// TIA Portal project "Process" (V16)

(* hardware
DEVICE "S7-1200 station_1"  S7-1200 Station
   slot 0: "Rack_0"  S7-1200 Rack  Rack  V1.0
   slot 1: "PLC_1"  CPU 1212C DC/DC/DC  6ES7 212-1AE40-0XB0  V4.4
   slot 2: "DI 8/DQ 8x24VDC_1"  6ES7 223-1BH32-0XB0  V2.0
   slot 3: "AI 4x13BIT/AQ 2x14BIT_1"  6ES7 234-4HE32-0XB0  V2.1
*)

// ===== PLC "PLC_1"  CPU 1212C DC/DC/DC =====

VAR_GLOBAL   // PLC tag table "Default tag table"
   "System_Byte" AT %MB1 : Byte;
   "FirstScan" AT %M1.0 : Bool;
   "DiagStatusUpdate" AT %M1.1 : Bool;
   "AlwaysTRUE" AT %M1.2 : Bool;
   "AlwaysFALSE" AT %M1.3 : Bool;
   "Clock_Byte" AT %MB0 : Byte;
   "Clock_10Hz" AT %M0.0 : Bool;
   "Clock_5Hz" AT %M0.1 : Bool;
   "Clock_2.5Hz" AT %M0.2 : Bool;
   "Clock_2Hz" AT %M0.3 : Bool;
   "Clock_1.25Hz" AT %M0.4 : Bool;
   "Clock_1Hz" AT %M0.5 : Bool;
   "Clock_0.625Hz" AT %M0.6 : Bool;
   "Clock_0.5Hz" AT %M0.7 : Bool;
END_VAR

VAR_GLOBAL   // PLC tag table "INPUTS"
   "FLD_IN_AD" AT %IW112 : Word;
   "FLD_IN_TERM" AT %IW114 : Word;
   "FLD_IN_RTD" AT %IW116 : Word;
END_VAR

DATA_BLOCK "OPC_EXC"   // DB1
{ S7_Optimized_Access := 'TRUE' }
VERSION : 0.1
   VAR
      TEMP_1 : Real;
      TEMP_2 : Real;
      TEMP_3 : Real;
      START_CAL : Bool;
   END_VAR
BEGIN
END_DATA_BLOCK

DATA_BLOCK "COMM"   // DB2
{ S7_Optimized_Access := 'TRUE' }
VERSION : 0.1
   VAR
      "counter" : UInt;
   END_VAR
BEGIN
END_DATA_BLOCK

FUNCTION "CALC_RTD_TEMP" : Void   // FC1, SCL
{ S7_Optimized_Access := 'TRUE' }
VERSION : 0.1
   VAR_INPUT
      IN_RAW : DInt;
      IN_VREF : Real;
      IN_R : Real;
   END_VAR
   VAR_OUTPUT
      CALC_RTD_TEMP : Real;
   END_VAR
   VAR_TEMP
      normalized : Real;
      voltage : Real;
      resistance : Real;
   END_VAR
   VAR CONSTANT
      alpha : Real := 0.00385;
      gamma : Real := 1.5;
      R_0 : Real := 100.0;
      "A" : Real := 0.00390775;
      "B" : Real := -5.77E-07;
   END_VAR
BEGIN
   #normalized := NORM_X(MIN := 0, VALUE := #IN_RAW, MAX := 27648);
   #voltage := SCALE_X(MIN:=0.0, VALUE:=#normalized, MAX:=10.0);
   #resistance := #voltage*#IN_R/(#IN_VREF-#voltage)-8.0;


   #CALC_RTD_TEMP := (- #A + SQRT(#A * #A - 4 * #B * (1 - #resistance / 100.0))) / (2 * #B);
END_FUNCTION

FUNCTION "CALC_LM_TEMP" : Void   // FC2, SCL
{ S7_Optimized_Access := 'TRUE' }
VERSION : 0.1
   VAR_INPUT
      IN_RAW : DInt;
      IN_FACTOR : Real;
   END_VAR
   VAR_OUTPUT
      CALC_AD_TEMP : Real;
   END_VAR
   VAR_TEMP
      normalized : Real;
      voltage : Real;
   END_VAR
BEGIN
   #normalized := NORM_X(MIN := 0, VALUE := #IN_RAW, MAX := 27648);
   #voltage := SCALE_X(MIN := 0.0, VALUE := #normalized, MAX := 10.0);


   #CALC_AD_TEMP := (#voltage/#IN_FACTOR);
END_FUNCTION

FUNCTION "CALC_TERM_TEMP" : Void   // FC3, SCL
{ S7_Optimized_Access := 'TRUE' }
VERSION : 0.1
   VAR_INPUT
      IN_RAW : DInt;
      IN_VREF : Real;
      IN_R : Real;
   END_VAR
   VAR_OUTPUT
      CALC_TERM_TEMP : Real;
   END_VAR
   VAR_TEMP
      normalized : Real;
      voltage : Real;
      resistance : Real;
      inv_temp : Real;
      ln_res : Real;
   END_VAR
   VAR CONSTANT
      "A" : Real := 0.001575561;
      "B" : Real := 0.0001422168;
      C : Real := 5.987E-07;
   END_VAR
BEGIN
   #normalized := NORM_X(MIN := 0, VALUE := #IN_RAW, MAX := 27648);
   #voltage := SCALE_X(MIN := 0.0, VALUE := #normalized, MAX := 10.0);
   #resistance := #voltage * #IN_R / (#IN_VREF - #voltage);

   #ln_res := LN(#resistance);
   #inv_temp := #A+#B*#ln_res+#C*#ln_res*#ln_res*#ln_res;

   #CALC_TERM_TEMP := 1/#inv_temp - 273.15;
END_FUNCTION

ORGANIZATION_BLOCK "Main"   // OB1, LAD, ProgramCycle
TITLE = "Main Program Sweep (Cycle)"
{ S7_Optimized_Access := 'TRUE' }
VERSION : 0.1
   VAR_INPUT
      Initial_Call : Bool;   // Initial call of this OB
      Remanence : Bool;   // =True, if remanent data are available
   END_VAR
BEGIN

REGION Network 1
   // Testing OPC UA
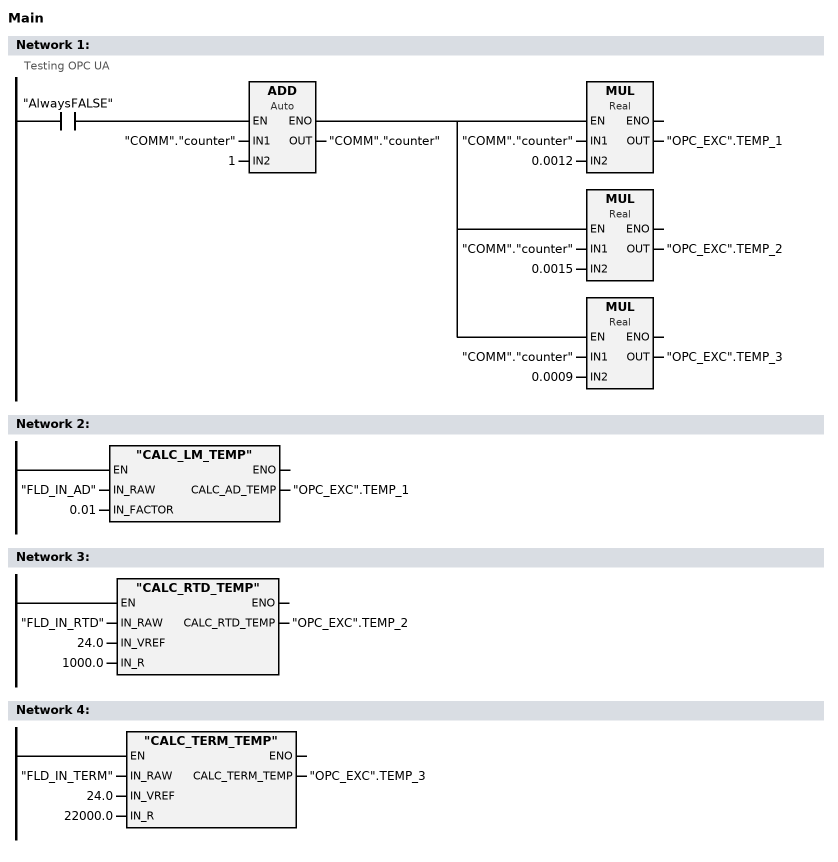
   RUNG wire#powerrail
      Contact( "AlwaysFALSE" )
      Add(in1 := "COMM"."counter", in2 := 1, out => "COMM"."counter")
      wire#w1
      { S7_Templates := "SrcType := Real" } Mul(in1 := "COMM"."counter", in2 := 0.0012, out => "OPC_EXC".TEMP_1)
   END_RUNG
   RUNG wire#w1
      { S7_Templates := "SrcType := Real" } Mul(in1 := "COMM"."counter", in2 := 0.0015, out => "OPC_EXC".TEMP_2)
   END_RUNG
   RUNG wire#w1
      { S7_Templates := "SrcType := Real" } Mul(in1 := "COMM"."counter", in2 := 0.0009, out => "OPC_EXC".TEMP_3)
   END_RUNG
   // the same network as SCL:
   IF "AlwaysFALSE" THEN
       "COMM"."counter" := "COMM"."counter" + 1;
       "OPC_EXC".TEMP_1 := "COMM"."counter" * 0.0012;
       "OPC_EXC".TEMP_2 := "COMM"."counter" * 0.0015;
       "OPC_EXC".TEMP_3 := "COMM"."counter" * 0.0009;
   END_IF;
END_REGION

REGION Network 2
   RUNG wire#powerrail
      "CALC_LM_TEMP"(IN_RAW := "FLD_IN_AD", IN_FACTOR := 0.01, CALC_AD_TEMP => "OPC_EXC".TEMP_1)
   END_RUNG
   // the same network as SCL:
   "CALC_LM_TEMP"(IN_RAW := "FLD_IN_AD", IN_FACTOR := 0.01, CALC_AD_TEMP => "OPC_EXC".TEMP_1);
END_REGION

REGION Network 3
   RUNG wire#powerrail
      "CALC_RTD_TEMP"(IN_RAW := "FLD_IN_RTD", IN_VREF := 24.0, IN_R := 1000.0, CALC_RTD_TEMP => "OPC_EXC".TEMP_2)
   END_RUNG
   // the same network as SCL:
   "CALC_RTD_TEMP"(IN_RAW := "FLD_IN_RTD", IN_VREF := 24.0, IN_R := 1000.0, CALC_RTD_TEMP => "OPC_EXC".TEMP_2);
END_REGION

REGION Network 4
   RUNG wire#powerrail
      "CALC_TERM_TEMP"(IN_RAW := "FLD_IN_TERM", IN_VREF := 24.0, IN_R := 22000.0, CALC_TERM_TEMP => "OPC_EXC".TEMP_3)
   END_RUNG
   // the same network as SCL:
   "CALC_TERM_TEMP"(IN_RAW := "FLD_IN_TERM",
                    IN_VREF := 24.0,
                    IN_R := 22000.0,
                    CALC_TERM_TEMP => "OPC_EXC".TEMP_3);
END_REGION
END_ORGANIZATION_BLOCK